(* IEC 61131-3 sources: CereveateHMI_Production_v2/CSharpBackend, 2 files *)

(* ---- FTP1_Simulation.st ---- *)
(* ============================================================
   FTP-1 POTLINE Simulation Program — FULL REPLACEMENT
   Auto-generated from Tag_master_Details_System_Upload.xlsx
   TOTAL TAGS: 128 (includes all 5 existing + 123 new)
   Set Sim_Enable := 1 to start, 0 to stop.
   Tags with NULL limits simulate within normal range only.
   All other tags oscillate across LL/HH -> triggers alarms.
   ============================================================ *)

VAR
    Sim_Enable  : BOOL := 0;

    (* --- Simulated tag variables --- *)
    PY1101A       : REAL := 1.16;
    Dir_PY1101A   : BOOL := 1;
    PY1101B       : REAL := 1.125;
    Dir_PY1101B   : BOOL := 1;
    PY1103A       : REAL := 17.45;
    Dir_PY1103A   : BOOL := 1;
    PY1103B       : REAL := 16.525;
    Dir_PY1103B   : BOOL := 1;
    TY1101A       : REAL := 59.4;
    Dir_TY1101A   : BOOL := 1;
    PY1104       : REAL := 7.35;
    Dir_PY1104   : BOOL := 1;
    PY1105A       : REAL := 0.405;
    Dir_PY1105A   : BOOL := 1;
    PY1105B       : REAL := 0.405;
    Dir_PY1105B   : BOOL := 1;
    PY1105C       : REAL := 0.405;
    Dir_PY1105C   : BOOL := 1;
    PY1105D       : REAL := 0.405;
    Dir_PY1105D   : BOOL := 1;
    PY1105E       : REAL := 0.405;
    Dir_PY1105E   : BOOL := 1;
    PY1105F       : REAL := 0.405;
    Dir_PY1105F   : BOOL := 1;
    PY1105G       : REAL := 0.405;
    Dir_PY1105G   : BOOL := 1;
    PY1105H       : REAL := 0.405;
    Dir_PY1105H   : BOOL := 1;
    PY1105I       : REAL := 0.405;
    Dir_PY1105I   : BOOL := 1;
    PY1105J       : REAL := 0.405;
    Dir_PY1105J   : BOOL := 1;
    TY1101B       : REAL := 75.0;
    Dir_TY1101B   : BOOL := 1;
    TY1101C       : REAL := 75.0;
    Dir_TY1101C   : BOOL := 1;
    TY1101D       : REAL := 75.0;
    Dir_TY1101D   : BOOL := 1;
    TY1101E       : REAL := 75.0;
    Dir_TY1101E   : BOOL := 1;
    TY1101F       : REAL := 75.0;
    Dir_TY1101F   : BOOL := 1;
    TY1101G       : REAL := 75.0;
    Dir_TY1101G   : BOOL := 1;
    TY1101H       : REAL := 75.0;
    Dir_TY1101H   : BOOL := 1;
    TY1102A       : REAL := 75.0;
    Dir_TY1102A   : BOOL := 1;
    TY1102B       : REAL := 75.0;
    Dir_TY1102B   : BOOL := 1;
    TY1102C       : REAL := 75.0;
    Dir_TY1102C   : BOOL := 1;
    TY1102D       : REAL := 75.0;
    Dir_TY1102D   : BOOL := 1;
    TY1102E       : REAL := 75.0;
    Dir_TY1102E   : BOOL := 1;
    TY1102F       : REAL := 75.0;
    Dir_TY1102F   : BOOL := 1;
    TY1102G       : REAL := 75.0;
    Dir_TY1102G   : BOOL := 1;
    TY1102H       : REAL := 75.0;
    Dir_TY1102H   : BOOL := 1;
    TY1103A       : REAL := 75.0;
    Dir_TY1103A   : BOOL := 1;
    TY1103B       : REAL := 75.0;
    Dir_TY1103B   : BOOL := 1;
    TY1103C       : REAL := 75.0;
    Dir_TY1103C   : BOOL := 1;
    TY1103D       : REAL := 75.0;
    Dir_TY1103D   : BOOL := 1;
    TY1103E       : REAL := 75.0;
    Dir_TY1103E   : BOOL := 1;
    TY1103F       : REAL := 75.0;
    Dir_TY1103F   : BOOL := 1;
    TY1103G       : REAL := 75.0;
    Dir_TY1103G   : BOOL := 1;
    TY1103H       : REAL := 75.0;
    Dir_TY1103H   : BOOL := 1;
    TY1104A       : REAL := 75.0;
    Dir_TY1104A   : BOOL := 1;
    TY1104B       : REAL := 75.0;
    Dir_TY1104B   : BOOL := 1;
    TY1104C       : REAL := 75.0;
    Dir_TY1104C   : BOOL := 1;
    TY1104D       : REAL := 75.0;
    Dir_TY1104D   : BOOL := 1;
    TY1104E       : REAL := 75.0;
    Dir_TY1104E   : BOOL := 1;
    TY1104F       : REAL := 75.0;
    Dir_TY1104F   : BOOL := 1;
    TY1104G       : REAL := 75.0;
    Dir_TY1104G   : BOOL := 1;
    TY1104H       : REAL := 75.0;
    Dir_TY1104H   : BOOL := 1;
    IYAN1101       : REAL := 45.0;
    Dir_IYAN1101   : BOOL := 1;
    IYAN1102       : REAL := 45.0;
    Dir_IYAN1102   : BOOL := 1;
    IYAN1103       : REAL := 45.0;
    Dir_IYAN1103   : BOOL := 1;
    IYAN1104       : REAL := 45.0;
    Dir_IYAN1104   : BOOL := 1;
    IYFBR1101       : REAL := 45.0;
    Dir_IYFBR1101   : BOOL := 1;
    IYFBR1102       : REAL := 45.0;
    Dir_IYFBR1102   : BOOL := 1;
    IYFBC1101       : REAL := 45.0;
    Dir_IYFBC1101   : BOOL := 1;
    IYFBC1102       : REAL := 45.0;
    Dir_IYFBC1102   : BOOL := 1;
    HZ1101A       : REAL := 50.0;
    Dir_HZ1101A   : BOOL := 1;
    HZ1102A       : REAL := 50.0;
    Dir_HZ1102A   : BOOL := 1;
    HZ1103A       : REAL := 50.0;
    Dir_HZ1103A   : BOOL := 1;
    HZ1104A       : REAL := 50.0;
    Dir_HZ1104A   : BOOL := 1;
    AY1101       : REAL := 42.5;
    Dir_AY1101   : BOOL := 1;
    AY1102       : REAL := 42.5;
    Dir_AY1102   : BOOL := 1;
    TY1105A       : REAL := 75.0;
    Dir_TY1105A   : BOOL := 1;
    TY1105B       : REAL := 75.0;
    Dir_TY1105B   : BOOL := 1;
    PDY1101       : REAL := 1.925;
    Dir_PDY1101   : BOOL := 1;
    PDY1102       : REAL := 1.925;
    Dir_PDY1102   : BOOL := 1;
    PDY1104       : REAL := 1.925;
    Dir_PDY1104   : BOOL := 1;
    PDY1105       : REAL := 1.925;
    Dir_PDY1105   : BOOL := 1;
    PDY1106A       : REAL := 1.925;
    Dir_PDY1106A   : BOOL := 1;
    PDY1107A       : REAL := 1.925;
    Dir_PDY1107A   : BOOL := 1;
    PDY1108       : REAL := 1.925;
    Dir_PDY1108   : BOOL := 1;
    PDY1109       : REAL := 1.925;
    Dir_PDY1109   : BOOL := 1;
    PDY1110       : REAL := 1.925;
    Dir_PDY1110   : BOOL := 1;
    FY1100       : REAL := 2250.0;
    Dir_FY1100   : BOOL := 1;
    VYAN1101A       : REAL := 3.75;
    Dir_VYAN1101A   : BOOL := 1;
    VYAN1101B       : REAL := 3.75;
    Dir_VYAN1101B   : BOOL := 1;
    VYAN1101C       : REAL := 3.75;
    Dir_VYAN1101C   : BOOL := 1;
    VYAN1101D       : REAL := 3.75;
    Dir_VYAN1101D   : BOOL := 1;
    VYAN1102A       : REAL := 3.75;
    Dir_VYAN1102A   : BOOL := 1;
    VYAN1102B       : REAL := 3.75;
    Dir_VYAN1102B   : BOOL := 1;
    VYAN1102C       : REAL := 3.75;
    Dir_VYAN1102C   : BOOL := 1;
    VYAN1102D       : REAL := 3.75;
    Dir_VYAN1102D   : BOOL := 1;
    VYAN1103A       : REAL := 3.75;
    Dir_VYAN1103A   : BOOL := 1;
    VYAN1103B       : REAL := 3.75;
    Dir_VYAN1103B   : BOOL := 1;
    VYAN1103C       : REAL := 3.75;
    Dir_VYAN1103C   : BOOL := 1;
    VYAN1103D       : REAL := 3.75;
    Dir_VYAN1103D   : BOOL := 1;
    VYAN1104A       : REAL := 3.75;
    Dir_VYAN1104A   : BOOL := 1;
    VYAN1104B       : REAL := 3.75;
    Dir_VYAN1104B   : BOOL := 1;
    VYAN1104C       : REAL := 3.75;
    Dir_VYAN1104C   : BOOL := 1;
    VYAN1104D       : REAL := 3.75;
    Dir_VYAN1104D   : BOOL := 1;
    PY1102A       : REAL := 22.5;
    Dir_PY1102A   : BOOL := 1;
    PY1102B       : REAL := 22.5;
    Dir_PY1102B   : BOOL := 1;
    PY1102C       : REAL := 22.5;
    Dir_PY1102C   : BOOL := 1;
    PY1102D       : REAL := 22.5;
    Dir_PY1102D   : BOOL := 1;
    LY3101       : REAL := 3.675;
    Dir_LY3101   : BOOL := 1;
    PY3101       : REAL := 1.925;
    Dir_PY3101   : BOOL := 1;
    LY1101       : REAL := 4.5;
    Dir_LY1101   : BOOL := 1;
    LY1102       : REAL := 4.5;
    Dir_LY1102   : BOOL := 1;
    FY3101       : REAL := 225.0;
    Dir_FY3101   : BOOL := 1;
    VY1101A       : REAL := 50.0;
    Dir_VY1101A   : BOOL := 1;
    FY1101       : REAL := 90.0;
    Dir_FY1101   : BOOL := 1;
    CV1101       : REAL := 52.5;
    Dir_CV1101   : BOOL := 1;
    TY3101       : REAL := 75.0;
    Dir_TY3101   : BOOL := 1;
    VYAN1101E       : REAL := 3.75;
    Dir_VYAN1101E   : BOOL := 1;
    VYAN1101F       : REAL := 3.75;
    Dir_VYAN1101F   : BOOL := 1;
    VYAN1101G       : REAL := 3.75;
    Dir_VYAN1101G   : BOOL := 1;
    VYAN1101H       : REAL := 3.75;
    Dir_VYAN1101H   : BOOL := 1;
    VYAN1102E       : REAL := 3.75;
    Dir_VYAN1102E   : BOOL := 1;
    VYAN1102F       : REAL := 3.75;
    Dir_VYAN1102F   : BOOL := 1;
    VYAN1102G       : REAL := 3.75;
    Dir_VYAN1102G   : BOOL := 1;
    VYAN1102H       : REAL := 3.75;
    Dir_VYAN1102H   : BOOL := 1;
    VYAN1103E       : REAL := 3.75;
    Dir_VYAN1103E   : BOOL := 1;
    VYAN1103F       : REAL := 3.75;
    Dir_VYAN1103F   : BOOL := 1;
    VYAN1103G       : REAL := 3.75;
    Dir_VYAN1103G   : BOOL := 1;
    VYAN1103H       : REAL := 3.75;
    Dir_VYAN1103H   : BOOL := 1;
    VYAN1104E       : REAL := 3.75;
    Dir_VYAN1104E   : BOOL := 1;
    VYAN1104F       : REAL := 3.75;
    Dir_VYAN1104F   : BOOL := 1;
    VYAN1104G       : REAL := 3.75;
    Dir_VYAN1104G   : BOOL := 1;
    VYAN1104H       : REAL := 3.75;
    Dir_VYAN1104H   : BOOL := 1;
    MV1101A       : REAL := 50.0;
    Dir_MV1101A   : BOOL := 1;
    MV1102A       : REAL := 50.0;
    Dir_MV1102A   : BOOL := 1;
    HZ1101B       : REAL := 50.0;
    Dir_HZ1101B   : BOOL := 1;
    HZ1102B       : REAL := 50.0;
    Dir_HZ1102B   : BOOL := 1;
    HZ1103B       : REAL := 50.0;
    Dir_HZ1103B   : BOOL := 1;
    HZ1104B       : REAL := 50.0;
    Dir_HZ1104B   : BOOL := 1;
    VT1101B       : REAL := 50.0;
    Dir_VT1101B   : BOOL := 1;
    CV1101B       : REAL := 52.5;
    Dir_CV1101B   : BOOL := 1;
    Fresh_SILO_MT       : REAL := 450.0;
    Dir_Fresh_SILO_MT   : BOOL := 1;
    Enrich_SILO_MT       : REAL := 450.0;
    Dir_Enrich_SILO_MT   : BOOL := 1;
END_VAR

(* ============================================================
   SIMULATION BODY
   ============================================================ *)
IF Sim_Enable THEN

    (* PY1101A - CHUTE SILO FAN OUTLET PRESSURE #1 [KPA] sim 0.48..1.84 *)
    IF Dir_PY1101A THEN
        PY1101A := PY1101A + 0.009067;
    ELSE
        PY1101A := PY1101A - 0.009067;
    END_IF;
    IF PY1101A >= 1.84 THEN Dir_PY1101A := 0; END_IF;
    IF PY1101A <= 0.48 THEN Dir_PY1101A := 1; END_IF;

    (* PY1101B - CHUTE SILO FAN OUTLET PRESSURE #2 [KPA] sim 0.64..1.61 *)
    IF Dir_PY1101B THEN
        PY1101B := PY1101B + 0.006467;
    ELSE
        PY1101B := PY1101B - 0.006467;
    END_IF;
    IF PY1101B >= 1.61 THEN Dir_PY1101B := 0; END_IF;
    IF PY1101B <= 0.64 THEN Dir_PY1101B := 1; END_IF;

    (* PY1103A - ID FAN OUTLET PRESSURE #1 [KPA] sim 9.6..25.3 *)
    IF Dir_PY1103A THEN
        PY1103A := PY1103A + 0.104667;
    ELSE
        PY1103A := PY1103A - 0.104667;
    END_IF;
    IF PY1103A >= 25.3 THEN Dir_PY1103A := 0; END_IF;
    IF PY1103A <= 9.6 THEN Dir_PY1103A := 1; END_IF;

    (* PY1103B - ID FAN OUTLET PRESSURE #2 [KPA] sim 11.2..21.85 *)
    IF Dir_PY1103B THEN
        PY1103B := PY1103B + 0.071;
    ELSE
        PY1103B := PY1103B - 0.071;
    END_IF;
    IF PY1103B >= 21.85 THEN Dir_PY1103B := 0; END_IF;
    IF PY1103B <= 11.2 THEN Dir_PY1103B := 1; END_IF;

    (* TY1101A - 1# ID FAN FRONT BEARING TEMPERATURE [°C] sim 36.0..82.8 *)
    IF Dir_TY1101A THEN
        TY1101A := TY1101A + 0.312;
    ELSE
        TY1101A := TY1101A - 0.312;
    END_IF;
    IF TY1101A >= 82.8 THEN Dir_TY1101A := 0; END_IF;
    IF TY1101A <= 36.0 THEN Dir_TY1101A := 1; END_IF;

    (* PY1104 - CHUTE  SILO FAN OUTLET OF PRESSURE [KPA] sim 3.2..11.5 *)
    IF Dir_PY1104 THEN
        PY1104 := PY1104 + 0.055333;
    ELSE
        PY1104 := PY1104 - 0.055333;
    END_IF;
    IF PY1104 >= 11.5 THEN Dir_PY1104 := 0; END_IF;
    IF PY1104 <= 3.2 THEN Dir_PY1104 := 1; END_IF;

    (* PY1105A - FILTER AIR BAG OF PRESSURE #1 [KPA] sim 0.12..0.69 *)
    IF Dir_PY1105A THEN
        PY1105A := PY1105A + 0.0038;
    ELSE
        PY1105A := PY1105A - 0.0038;
    END_IF;
    IF PY1105A >= 0.69 THEN Dir_PY1105A := 0; END_IF;
    IF PY1105A <= 0.12 THEN Dir_PY1105A := 1; END_IF;

    (* PY1105B - FILTER AIR BAG OF PRESSURE #2 [KPA] sim 0.12..0.69 *)
    IF Dir_PY1105B THEN
        PY1105B := PY1105B + 0.0038;
    ELSE
        PY1105B := PY1105B - 0.0038;
    END_IF;
    IF PY1105B >= 0.69 THEN Dir_PY1105B := 0; END_IF;
    IF PY1105B <= 0.12 THEN Dir_PY1105B := 1; END_IF;

    (* PY1105C - FILTER AIR BAG OF PRESSURE #3 [KPA] sim 0.12..0.69 *)
    IF Dir_PY1105C THEN
        PY1105C := PY1105C + 0.0038;
    ELSE
        PY1105C := PY1105C - 0.0038;
    END_IF;
    IF PY1105C >= 0.69 THEN Dir_PY1105C := 0; END_IF;
    IF PY1105C <= 0.12 THEN Dir_PY1105C := 1; END_IF;

    (* PY1105D - FILTER AIR BAG OF PRESSURE #4 [KPA] sim 0.12..0.69 *)
    IF Dir_PY1105D THEN
        PY1105D := PY1105D + 0.0038;
    ELSE
        PY1105D := PY1105D - 0.0038;
    END_IF;
    IF PY1105D >= 0.69 THEN Dir_PY1105D := 0; END_IF;
    IF PY1105D <= 0.12 THEN Dir_PY1105D := 1; END_IF;

    (* PY1105E - FILTER AIR BAG OF PRESSURE #5 [KPA] sim 0.12..0.69 *)
    IF Dir_PY1105E THEN
        PY1105E := PY1105E + 0.0038;
    ELSE
        PY1105E := PY1105E - 0.0038;
    END_IF;
    IF PY1105E >= 0.69 THEN Dir_PY1105E := 0; END_IF;
    IF PY1105E <= 0.12 THEN Dir_PY1105E := 1; END_IF;

    (* PY1105F - FILTER AIR BAG OF PRESSURE #6 [KPA] sim 0.12..0.69 *)
    IF Dir_PY1105F THEN
        PY1105F := PY1105F + 0.0038;
    ELSE
        PY1105F := PY1105F - 0.0038;
    END_IF;
    IF PY1105F >= 0.69 THEN Dir_PY1105F := 0; END_IF;
    IF PY1105F <= 0.12 THEN Dir_PY1105F := 1; END_IF;

    (* PY1105G - FILTER AIR BAG OF PRESSURE #7 [KPA] sim 0.12..0.69 *)
    IF Dir_PY1105G THEN
        PY1105G := PY1105G + 0.0038;
    ELSE
        PY1105G := PY1105G - 0.0038;
    END_IF;
    IF PY1105G >= 0.69 THEN Dir_PY1105G := 0; END_IF;
    IF PY1105G <= 0.12 THEN Dir_PY1105G := 1; END_IF;

    (* PY1105H - FILTER AIR BAG OF PRESSURE #8 [KPA] sim 0.12..0.69 *)
    IF Dir_PY1105H THEN
        PY1105H := PY1105H + 0.0038;
    ELSE
        PY1105H := PY1105H - 0.0038;
    END_IF;
    IF PY1105H >= 0.69 THEN Dir_PY1105H := 0; END_IF;
    IF PY1105H <= 0.12 THEN Dir_PY1105H := 1; END_IF;

    (* PY1105I - FILTER AIR BAG OF PRESSURE #9 [KPA] sim 0.12..0.69 *)
    IF Dir_PY1105I THEN
        PY1105I := PY1105I + 0.0038;
    ELSE
        PY1105I := PY1105I - 0.0038;
    END_IF;
    IF PY1105I >= 0.69 THEN Dir_PY1105I := 0; END_IF;
    IF PY1105I <= 0.12 THEN Dir_PY1105I := 1; END_IF;

    (* PY1105J - FILTER AIR BAG OF PRESSURE #10 [KPA] sim 0.12..0.69 *)
    IF Dir_PY1105J THEN
        PY1105J := PY1105J + 0.0038;
    ELSE
        PY1105J := PY1105J - 0.0038;
    END_IF;
    IF PY1105J >= 0.69 THEN Dir_PY1105J := 0; END_IF;
    IF PY1105J <= 0.12 THEN Dir_PY1105J := 1; END_IF;

    (* TY1101B - 1# ID FAN REAR BEARING TEMPERATURE [°C] sim 30.0..120.0 *)
    IF Dir_TY1101B THEN
        TY1101B := TY1101B + 0.6;
    ELSE
        TY1101B := TY1101B - 0.6;
    END_IF;
    IF TY1101B >= 120.0 THEN Dir_TY1101B := 0; END_IF;
    IF TY1101B <= 30.0 THEN Dir_TY1101B := 1; END_IF;

    (* TY1101C - 1# ID FAN MOTOR FRONT BEARING TEMPERATURE [°C] sim 30.0..120.0 *)
    IF Dir_TY1101C THEN
        TY1101C := TY1101C + 0.6;
    ELSE
        TY1101C := TY1101C - 0.6;
    END_IF;
    IF TY1101C >= 120.0 THEN Dir_TY1101C := 0; END_IF;
    IF TY1101C <= 30.0 THEN Dir_TY1101C := 1; END_IF;

    (* TY1101D - 1# ID FAN MOTOR REAR BEARING TEMPERATURE [°C] sim 30.0..120.0 *)
    IF Dir_TY1101D THEN
        TY1101D := TY1101D + 0.6;
    ELSE
        TY1101D := TY1101D - 0.6;
    END_IF;
    IF TY1101D >= 120.0 THEN Dir_TY1101D := 0; END_IF;
    IF TY1101D <= 30.0 THEN Dir_TY1101D := 1; END_IF;

    (* TY1101E - 1# ID FAN  MOTOR Winding temperature A [°C] sim 30.0..120.0 *)
    IF Dir_TY1101E THEN
        TY1101E := TY1101E + 0.6;
    ELSE
        TY1101E := TY1101E - 0.6;
    END_IF;
    IF TY1101E >= 120.0 THEN Dir_TY1101E := 0; END_IF;
    IF TY1101E <= 30.0 THEN Dir_TY1101E := 1; END_IF;

    (* TY1101F - 1# ID FAN  MOTOR Winding temperature B [°C] sim 30.0..120.0 *)
    IF Dir_TY1101F THEN
        TY1101F := TY1101F + 0.6;
    ELSE
        TY1101F := TY1101F - 0.6;
    END_IF;
    IF TY1101F >= 120.0 THEN Dir_TY1101F := 0; END_IF;
    IF TY1101F <= 30.0 THEN Dir_TY1101F := 1; END_IF;

    (* TY1101G - 1# ID FAN  MOTOR Winding temperature C [°C] sim 30.0..120.0 *)
    IF Dir_TY1101G THEN
        TY1101G := TY1101G + 0.6;
    ELSE
        TY1101G := TY1101G - 0.6;
    END_IF;
    IF TY1101G >= 120.0 THEN Dir_TY1101G := 0; END_IF;
    IF TY1101G <= 30.0 THEN Dir_TY1101G := 1; END_IF;

    (* TY1101H - 1# ID FAN INLET TEMPERATURE [°C] sim 30.0..120.0 *)
    IF Dir_TY1101H THEN
        TY1101H := TY1101H + 0.6;
    ELSE
        TY1101H := TY1101H - 0.6;
    END_IF;
    IF TY1101H >= 120.0 THEN Dir_TY1101H := 0; END_IF;
    IF TY1101H <= 30.0 THEN Dir_TY1101H := 1; END_IF;

    (* TY1102A - 2# ID FAN FRONT BEARING TEMPERATURE [°C] sim 30.0..120.0 *)
    IF Dir_TY1102A THEN
        TY1102A := TY1102A + 0.6;
    ELSE
        TY1102A := TY1102A - 0.6;
    END_IF;
    IF TY1102A >= 120.0 THEN Dir_TY1102A := 0; END_IF;
    IF TY1102A <= 30.0 THEN Dir_TY1102A := 1; END_IF;

    (* TY1102B - 2# ID FAN REAR BEARING TEMPERATURE [°C] sim 30.0..120.0 *)
    IF Dir_TY1102B THEN
        TY1102B := TY1102B + 0.6;
    ELSE
        TY1102B := TY1102B - 0.6;
    END_IF;
    IF TY1102B >= 120.0 THEN Dir_TY1102B := 0; END_IF;
    IF TY1102B <= 30.0 THEN Dir_TY1102B := 1; END_IF;

    (* TY1102C - 2# ID FAN MOTOR FRONT BEARING TEMPERATURE [°C] sim 30.0..120.0 *)
    IF Dir_TY1102C THEN
        TY1102C := TY1102C + 0.6;
    ELSE
        TY1102C := TY1102C - 0.6;
    END_IF;
    IF TY1102C >= 120.0 THEN Dir_TY1102C := 0; END_IF;
    IF TY1102C <= 30.0 THEN Dir_TY1102C := 1; END_IF;

    (* TY1102D - 2# ID FAN MOTOR REAR BEARING TEMPERATURE [°C] sim 30.0..120.0 *)
    IF Dir_TY1102D THEN
        TY1102D := TY1102D + 0.6;
    ELSE
        TY1102D := TY1102D - 0.6;
    END_IF;
    IF TY1102D >= 120.0 THEN Dir_TY1102D := 0; END_IF;
    IF TY1102D <= 30.0 THEN Dir_TY1102D := 1; END_IF;

    (* TY1102E - 2# ID FAN  MOTOR Winding temperature A [°C] sim 30.0..120.0 *)
    IF Dir_TY1102E THEN
        TY1102E := TY1102E + 0.6;
    ELSE
        TY1102E := TY1102E - 0.6;
    END_IF;
    IF TY1102E >= 120.0 THEN Dir_TY1102E := 0; END_IF;
    IF TY1102E <= 30.0 THEN Dir_TY1102E := 1; END_IF;

    (* TY1102F - 2# ID FAN  MOTOR Winding temperature B [°C] sim 30.0..120.0 *)
    IF Dir_TY1102F THEN
        TY1102F := TY1102F + 0.6;
    ELSE
        TY1102F := TY1102F - 0.6;
    END_IF;
    IF TY1102F >= 120.0 THEN Dir_TY1102F := 0; END_IF;
    IF TY1102F <= 30.0 THEN Dir_TY1102F := 1; END_IF;

    (* TY1102G - 2# ID FAN  MOTOR Winding temperature C [°C] sim 30.0..120.0 *)
    IF Dir_TY1102G THEN
        TY1102G := TY1102G + 0.6;
    ELSE
        TY1102G := TY1102G - 0.6;
    END_IF;
    IF TY1102G >= 120.0 THEN Dir_TY1102G := 0; END_IF;
    IF TY1102G <= 30.0 THEN Dir_TY1102G := 1; END_IF;

    (* TY1102H - 2# ID FAN INLET TEMPERATURE [°C] sim 30.0..120.0 *)
    IF Dir_TY1102H THEN
        TY1102H := TY1102H + 0.6;
    ELSE
        TY1102H := TY1102H - 0.6;
    END_IF;
    IF TY1102H >= 120.0 THEN Dir_TY1102H := 0; END_IF;
    IF TY1102H <= 30.0 THEN Dir_TY1102H := 1; END_IF;

    (* TY1103A - 3# ID FAN FRONT BEARING TEMPERATURE [°C] sim 30.0..120.0 *)
    IF Dir_TY1103A THEN
        TY1103A := TY1103A + 0.6;
    ELSE
        TY1103A := TY1103A - 0.6;
    END_IF;
    IF TY1103A >= 120.0 THEN Dir_TY1103A := 0; END_IF;
    IF TY1103A <= 30.0 THEN Dir_TY1103A := 1; END_IF;

    (* TY1103B - 3# ID FAN REAR BEARING TEMPERATURE [°C] sim 30.0..120.0 *)
    IF Dir_TY1103B THEN
        TY1103B := TY1103B + 0.6;
    ELSE
        TY1103B := TY1103B - 0.6;
    END_IF;
    IF TY1103B >= 120.0 THEN Dir_TY1103B := 0; END_IF;
    IF TY1103B <= 30.0 THEN Dir_TY1103B := 1; END_IF;

    (* TY1103C - 3# ID FAN MOTOR FRONT BEARING TEMPERATURE [°C] sim 30.0..120.0 *)
    IF Dir_TY1103C THEN
        TY1103C := TY1103C + 0.6;
    ELSE
        TY1103C := TY1103C - 0.6;
    END_IF;
    IF TY1103C >= 120.0 THEN Dir_TY1103C := 0; END_IF;
    IF TY1103C <= 30.0 THEN Dir_TY1103C := 1; END_IF;

    (* TY1103D - 3# ID FAN MOTOR REAR BEARING TEMPERATURE [°C] sim 30.0..120.0 *)
    IF Dir_TY1103D THEN
        TY1103D := TY1103D + 0.6;
    ELSE
        TY1103D := TY1103D - 0.6;
    END_IF;
    IF TY1103D >= 120.0 THEN Dir_TY1103D := 0; END_IF;
    IF TY1103D <= 30.0 THEN Dir_TY1103D := 1; END_IF;

    (* TY1103E - 3# ID FAN  MOTOR Winding temperature A [°C] sim 30.0..120.0 *)
    IF Dir_TY1103E THEN
        TY1103E := TY1103E + 0.6;
    ELSE
        TY1103E := TY1103E - 0.6;
    END_IF;
    IF TY1103E >= 120.0 THEN Dir_TY1103E := 0; END_IF;
    IF TY1103E <= 30.0 THEN Dir_TY1103E := 1; END_IF;

    (* TY1103F - 3# ID FAN  MOTOR Winding temperature B [°C] sim 30.0..120.0 *)
    IF Dir_TY1103F THEN
        TY1103F := TY1103F + 0.6;
    ELSE
        TY1103F := TY1103F - 0.6;
    END_IF;
    IF TY1103F >= 120.0 THEN Dir_TY1103F := 0; END_IF;
    IF TY1103F <= 30.0 THEN Dir_TY1103F := 1; END_IF;

    (* TY1103G - 3# ID FAN  MOTOR Winding temperature C [°C] sim 30.0..120.0 *)
    IF Dir_TY1103G THEN
        TY1103G := TY1103G + 0.6;
    ELSE
        TY1103G := TY1103G - 0.6;
    END_IF;
    IF TY1103G >= 120.0 THEN Dir_TY1103G := 0; END_IF;
    IF TY1103G <= 30.0 THEN Dir_TY1103G := 1; END_IF;

    (* TY1103H - 3# ID FAN INLET TEMPERATURE [°C] sim 30.0..120.0 *)
    IF Dir_TY1103H THEN
        TY1103H := TY1103H + 0.6;
    ELSE
        TY1103H := TY1103H - 0.6;
    END_IF;
    IF TY1103H >= 120.0 THEN Dir_TY1103H := 0; END_IF;
    IF TY1103H <= 30.0 THEN Dir_TY1103H := 1; END_IF;

    (* TY1104A - 4# ID FAN FRONT BEARING TEMPERATURE [°C] sim 30.0..120.0 *)
    IF Dir_TY1104A THEN
        TY1104A := TY1104A + 0.6;
    ELSE
        TY1104A := TY1104A - 0.6;
    END_IF;
    IF TY1104A >= 120.0 THEN Dir_TY1104A := 0; END_IF;
    IF TY1104A <= 30.0 THEN Dir_TY1104A := 1; END_IF;

    (* TY1104B - 4# ID FAN REAR BEARING TEMPERATURE [°C] sim 30.0..120.0 *)
    IF Dir_TY1104B THEN
        TY1104B := TY1104B + 0.6;
    ELSE
        TY1104B := TY1104B - 0.6;
    END_IF;
    IF TY1104B >= 120.0 THEN Dir_TY1104B := 0; END_IF;
    IF TY1104B <= 30.0 THEN Dir_TY1104B := 1; END_IF;

    (* TY1104C - 4# ID FAN MOTOR FRONT BEARING TEMPERATURE [°C] sim 30.0..120.0 *)
    IF Dir_TY1104C THEN
        TY1104C := TY1104C + 0.6;
    ELSE
        TY1104C := TY1104C - 0.6;
    END_IF;
    IF TY1104C >= 120.0 THEN Dir_TY1104C := 0; END_IF;
    IF TY1104C <= 30.0 THEN Dir_TY1104C := 1; END_IF;

    (* TY1104D - 4# ID FAN MOTOR REAR BEARING TEMPERATURE [°C] sim 30.0..120.0 *)
    IF Dir_TY1104D THEN
        TY1104D := TY1104D + 0.6;
    ELSE
        TY1104D := TY1104D - 0.6;
    END_IF;
    IF TY1104D >= 120.0 THEN Dir_TY1104D := 0; END_IF;
    IF TY1104D <= 30.0 THEN Dir_TY1104D := 1; END_IF;

    (* TY1104E - 4# ID FAN  MOTOR Winding temperature A [°C] sim 30.0..120.0 *)
    IF Dir_TY1104E THEN
        TY1104E := TY1104E + 0.6;
    ELSE
        TY1104E := TY1104E - 0.6;
    END_IF;
    IF TY1104E >= 120.0 THEN Dir_TY1104E := 0; END_IF;
    IF TY1104E <= 30.0 THEN Dir_TY1104E := 1; END_IF;

    (* TY1104F - 4# ID FAN  MOTOR Winding temperature B [°C] sim 30.0..120.0 *)
    IF Dir_TY1104F THEN
        TY1104F := TY1104F + 0.6;
    ELSE
        TY1104F := TY1104F - 0.6;
    END_IF;
    IF TY1104F >= 120.0 THEN Dir_TY1104F := 0; END_IF;
    IF TY1104F <= 30.0 THEN Dir_TY1104F := 1; END_IF;

    (* TY1104G - 4# ID FAN  MOTOR Winding temperature C [°C] sim 30.0..120.0 *)
    IF Dir_TY1104G THEN
        TY1104G := TY1104G + 0.6;
    ELSE
        TY1104G := TY1104G - 0.6;
    END_IF;
    IF TY1104G >= 120.0 THEN Dir_TY1104G := 0; END_IF;
    IF TY1104G <= 30.0 THEN Dir_TY1104G := 1; END_IF;

    (* TY1104H - 4# ID FAN INLET TEMPERATURE [°C] sim 30.0..120.0 *)
    IF Dir_TY1104H THEN
        TY1104H := TY1104H + 0.6;
    ELSE
        TY1104H := TY1104H - 0.6;
    END_IF;
    IF TY1104H >= 120.0 THEN Dir_TY1104H := 0; END_IF;
    IF TY1104H <= 30.0 THEN Dir_TY1104H := 1; END_IF;

    (* IYAN1101 - ID FAN CURRENT #1 [Amp] sim 10.0..80.0 *)
    IF Dir_IYAN1101 THEN
        IYAN1101 := IYAN1101 + 0.466667;
    ELSE
        IYAN1101 := IYAN1101 - 0.466667;
    END_IF;
    IF IYAN1101 >= 80.0 THEN Dir_IYAN1101 := 0; END_IF;
    IF IYAN1101 <= 10.0 THEN Dir_IYAN1101 := 1; END_IF;

    (* IYAN1102 - ID FAN CURRENT #2 [Amp] sim 10.0..80.0 *)
    IF Dir_IYAN1102 THEN
        IYAN1102 := IYAN1102 + 0.466667;
    ELSE
        IYAN1102 := IYAN1102 - 0.466667;
    END_IF;
    IF IYAN1102 >= 80.0 THEN Dir_IYAN1102 := 0; END_IF;
    IF IYAN1102 <= 10.0 THEN Dir_IYAN1102 := 1; END_IF;

    (* IYAN1103 - ID FAN CURRENT #3 [Amp] sim 10.0..80.0 *)
    IF Dir_IYAN1103 THEN
        IYAN1103 := IYAN1103 + 0.466667;
    ELSE
        IYAN1103 := IYAN1103 - 0.466667;
    END_IF;
    IF IYAN1103 >= 80.0 THEN Dir_IYAN1103 := 0; END_IF;
    IF IYAN1103 <= 10.0 THEN Dir_IYAN1103 := 1; END_IF;

    (* IYAN1104 - ID FAN CURRENT #4 [Amp] sim 10.0..80.0 *)
    IF Dir_IYAN1104 THEN
        IYAN1104 := IYAN1104 + 0.466667;
    ELSE
        IYAN1104 := IYAN1104 - 0.466667;
    END_IF;
    IF IYAN1104 >= 80.0 THEN Dir_IYAN1104 := 0; END_IF;
    IF IYAN1104 <= 10.0 THEN Dir_IYAN1104 := 1; END_IF;

    (* IYFBR1101 - ROOTS FAN CURRENT #1 [Amp] sim 10.0..80.0 *)
    IF Dir_IYFBR1101 THEN
        IYFBR1101 := IYFBR1101 + 0.466667;
    ELSE
        IYFBR1101 := IYFBR1101 - 0.466667;
    END_IF;
    IF IYFBR1101 >= 80.0 THEN Dir_IYFBR1101 := 0; END_IF;
    IF IYFBR1101 <= 10.0 THEN Dir_IYFBR1101 := 1; END_IF;

    (* IYFBR1102 - ROOTS FAN CURRENT #2 [Amp] sim 10.0..80.0 *)
    IF Dir_IYFBR1102 THEN
        IYFBR1102 := IYFBR1102 + 0.466667;
    ELSE
        IYFBR1102 := IYFBR1102 - 0.466667;
    END_IF;
    IF IYFBR1102 >= 80.0 THEN Dir_IYFBR1102 := 0; END_IF;
    IF IYFBR1102 <= 10.0 THEN Dir_IYFBR1102 := 1; END_IF;

    (* IYFBC1101 - HIGHT PRESSURE CENTRIFUGAL VENTILATOR #1 [Amp] sim 10.0..80.0 *)
    IF Dir_IYFBC1101 THEN
        IYFBC1101 := IYFBC1101 + 0.466667;
    ELSE
        IYFBC1101 := IYFBC1101 - 0.466667;
    END_IF;
    IF IYFBC1101 >= 80.0 THEN Dir_IYFBC1101 := 0; END_IF;
    IF IYFBC1101 <= 10.0 THEN Dir_IYFBC1101 := 1; END_IF;

    (* IYFBC1102 - HIGHT PRESSURE CENTRIFUGAL VENTILATOR #2 [Amp] sim 10.0..80.0 *)
    IF Dir_IYFBC1102 THEN
        IYFBC1102 := IYFBC1102 + 0.466667;
    ELSE
        IYFBC1102 := IYFBC1102 - 0.466667;
    END_IF;
    IF IYFBC1102 >= 80.0 THEN Dir_IYFBC1102 := 0; END_IF;
    IF IYFBC1102 <= 10.0 THEN Dir_IYFBC1102 := 1; END_IF;

    (* HZ1101A - ID FAN VALVE OF DEGREE (DAMPER FEEDBACK) #1 [%] sim 20.0..80.0 *)
    IF Dir_HZ1101A THEN
        HZ1101A := HZ1101A + 0.4;
    ELSE
        HZ1101A := HZ1101A - 0.4;
    END_IF;
    IF HZ1101A >= 80.0 THEN Dir_HZ1101A := 0; END_IF;
    IF HZ1101A <= 20.0 THEN Dir_HZ1101A := 1; END_IF;

    (* HZ1102A - ID FAN VALVE OF DEGREE (DAMPER FEEDBACK) #2 [%] sim 20.0..80.0 *)
    IF Dir_HZ1102A THEN
        HZ1102A := HZ1102A + 0.4;
    ELSE
        HZ1102A := HZ1102A - 0.4;
    END_IF;
    IF HZ1102A >= 80.0 THEN Dir_HZ1102A := 0; END_IF;
    IF HZ1102A <= 20.0 THEN Dir_HZ1102A := 1; END_IF;

    (* HZ1103A - ID FAN VALVE OF DEGREE (DAMPER FEEDBACK) #3 [%] sim 20.0..80.0 *)
    IF Dir_HZ1103A THEN
        HZ1103A := HZ1103A + 0.4;
    ELSE
        HZ1103A := HZ1103A - 0.4;
    END_IF;
    IF HZ1103A >= 80.0 THEN Dir_HZ1103A := 0; END_IF;
    IF HZ1103A <= 20.0 THEN Dir_HZ1103A := 1; END_IF;

    (* HZ1104A - ID FAN VALVE OF DEGREE (DAMPER FEEDBACK) #4 [%] sim 20.0..80.0 *)
    IF Dir_HZ1104A THEN
        HZ1104A := HZ1104A + 0.4;
    ELSE
        HZ1104A := HZ1104A - 0.4;
    END_IF;
    IF HZ1104A >= 80.0 THEN Dir_HZ1104A := 0; END_IF;
    IF HZ1104A <= 20.0 THEN Dir_HZ1104A := 1; END_IF;

    (* AY1101 - FTP-1 DUST ANALYZER [mg/m3] sim 5.0..80.0 *)
    IF Dir_AY1101 THEN
        AY1101 := AY1101 + 0.5;
    ELSE
        AY1101 := AY1101 - 0.5;
    END_IF;
    IF AY1101 >= 80.0 THEN Dir_AY1101 := 0; END_IF;
    IF AY1101 <= 5.0 THEN Dir_AY1101 := 1; END_IF;

    (* AY1102 - FTP-1 HF ANALYZER [mg/m3] sim 5.0..80.0 *)
    IF Dir_AY1102 THEN
        AY1102 := AY1102 + 0.5;
    ELSE
        AY1102 := AY1102 - 0.5;
    END_IF;
    IF AY1102 >= 80.0 THEN Dir_AY1102 := 0; END_IF;
    IF AY1102 <= 5.0 THEN Dir_AY1102 := 1; END_IF;

    (* TY1105A - FILTER INLET TEMPERATURE #1 [°C] sim 30.0..120.0 *)
    IF Dir_TY1105A THEN
        TY1105A := TY1105A + 0.6;
    ELSE
        TY1105A := TY1105A - 0.6;
    END_IF;
    IF TY1105A >= 120.0 THEN Dir_TY1105A := 0; END_IF;
    IF TY1105A <= 30.0 THEN Dir_TY1105A := 1; END_IF;

    (* TY1105B - FILTER INLET TEMPERATURE #2 [°C] sim 30.0..120.0 *)
    IF Dir_TY1105B THEN
        TY1105B := TY1105B + 0.6;
    ELSE
        TY1105B := TY1105B - 0.6;
    END_IF;
    IF TY1105B >= 120.0 THEN Dir_TY1105B := 0; END_IF;
    IF TY1105B <= 30.0 THEN Dir_TY1105B := 1; END_IF;

    (* PDY1101 - FILTER INLET  OUTLET PRESSURE #1 [KPA] sim 0.4..3.45 *)
    IF Dir_PDY1101 THEN
        PDY1101 := PDY1101 + 0.020333;
    ELSE
        PDY1101 := PDY1101 - 0.020333;
    END_IF;
    IF PDY1101 >= 3.45 THEN Dir_PDY1101 := 0; END_IF;
    IF PDY1101 <= 0.4 THEN Dir_PDY1101 := 1; END_IF;

    (* PDY1102 - FILTER INLET  OUTLET PRESSURE #2 [KPA] sim 0.4..3.45 *)
    IF Dir_PDY1102 THEN
        PDY1102 := PDY1102 + 0.020333;
    ELSE
        PDY1102 := PDY1102 - 0.020333;
    END_IF;
    IF PDY1102 >= 3.45 THEN Dir_PDY1102 := 0; END_IF;
    IF PDY1102 <= 0.4 THEN Dir_PDY1102 := 1; END_IF;

    (* PDY1104 - FILTER INLET  OUTLET PRESSURE #4 [KPA] sim 0.4..3.45 *)
    IF Dir_PDY1104 THEN
        PDY1104 := PDY1104 + 0.020333;
    ELSE
        PDY1104 := PDY1104 - 0.020333;
    END_IF;
    IF PDY1104 >= 3.45 THEN Dir_PDY1104 := 0; END_IF;
    IF PDY1104 <= 0.4 THEN Dir_PDY1104 := 1; END_IF;

    (* PDY1105 - FILTER INLET  OUTLET PRESSURE #5 [KPA] sim 0.4..3.45 *)
    IF Dir_PDY1105 THEN
        PDY1105 := PDY1105 + 0.020333;
    ELSE
        PDY1105 := PDY1105 - 0.020333;
    END_IF;
    IF PDY1105 >= 3.45 THEN Dir_PDY1105 := 0; END_IF;
    IF PDY1105 <= 0.4 THEN Dir_PDY1105 := 1; END_IF;

    (* PDY1106A - FILTER INLET  OUTLET PRESSURE #6 [KPA] sim 0.4..3.45 *)
    IF Dir_PDY1106A THEN
        PDY1106A := PDY1106A + 0.020333;
    ELSE
        PDY1106A := PDY1106A - 0.020333;
    END_IF;
    IF PDY1106A >= 3.45 THEN Dir_PDY1106A := 0; END_IF;
    IF PDY1106A <= 0.4 THEN Dir_PDY1106A := 1; END_IF;

    (* PDY1107A - FILTER INLET  OUTLET PRESSURE #7 [KPA] sim 0.4..3.45 *)
    IF Dir_PDY1107A THEN
        PDY1107A := PDY1107A + 0.020333;
    ELSE
        PDY1107A := PDY1107A - 0.020333;
    END_IF;
    IF PDY1107A >= 3.45 THEN Dir_PDY1107A := 0; END_IF;
    IF PDY1107A <= 0.4 THEN Dir_PDY1107A := 1; END_IF;

    (* PDY1108 - FILTER INLET  OUTLET PRESSURE #8 [KPA] sim 0.4..3.45 *)
    IF Dir_PDY1108 THEN
        PDY1108 := PDY1108 + 0.020333;
    ELSE
        PDY1108 := PDY1108 - 0.020333;
    END_IF;
    IF PDY1108 >= 3.45 THEN Dir_PDY1108 := 0; END_IF;
    IF PDY1108 <= 0.4 THEN Dir_PDY1108 := 1; END_IF;

    (* PDY1109 - FILTER INLET  OUTLET PRESSURE #9 [KPA] sim 0.4..3.45 *)
    IF Dir_PDY1109 THEN
        PDY1109 := PDY1109 + 0.020333;
    ELSE
        PDY1109 := PDY1109 - 0.020333;
    END_IF;
    IF PDY1109 >= 3.45 THEN Dir_PDY1109 := 0; END_IF;
    IF PDY1109 <= 0.4 THEN Dir_PDY1109 := 1; END_IF;

    (* PDY1110 - FILTER INLET  OUTLET PRESSURE #10 [KPA] sim 0.4..3.45 *)
    IF Dir_PDY1110 THEN
        PDY1110 := PDY1110 + 0.020333;
    ELSE
        PDY1110 := PDY1110 - 0.020333;
    END_IF;
    IF PDY1110 >= 3.45 THEN Dir_PDY1110 := 0; END_IF;
    IF PDY1110 <= 0.4 THEN Dir_PDY1110 := 1; END_IF;

    (* FY1100 - OUTLET FLOW [Nm3/Hr] sim 500.0..4000.0 *)
    IF Dir_FY1100 THEN
        FY1100 := FY1100 + 23.333333;
    ELSE
        FY1100 := FY1100 - 23.333333;
    END_IF;
    IF FY1100 >= 4000.0 THEN Dir_FY1100 := 0; END_IF;
    IF FY1100 <= 500.0 THEN Dir_FY1100 := 1; END_IF;

    (* VYAN1101A - ID FAN FRONT BEARING X VIBRATION #1 [mm/s] sim 0.5..7.0 *)
    IF Dir_VYAN1101A THEN
        VYAN1101A := VYAN1101A + 0.043333;
    ELSE
        VYAN1101A := VYAN1101A - 0.043333;
    END_IF;
    IF VYAN1101A >= 7.0 THEN Dir_VYAN1101A := 0; END_IF;
    IF VYAN1101A <= 0.5 THEN Dir_VYAN1101A := 1; END_IF;

    (* VYAN1101B - ID FAN FRONT BEARING Y VIBRATION #1 [mm/s] sim 0.5..7.0 *)
    IF Dir_VYAN1101B THEN
        VYAN1101B := VYAN1101B + 0.043333;
    ELSE
        VYAN1101B := VYAN1101B - 0.043333;
    END_IF;
    IF VYAN1101B >= 7.0 THEN Dir_VYAN1101B := 0; END_IF;
    IF VYAN1101B <= 0.5 THEN Dir_VYAN1101B := 1; END_IF;

    (* VYAN1101C - ID FAN REAR BEARING X VIBRATION #1 [mm/s] sim 0.5..7.0 *)
    IF Dir_VYAN1101C THEN
        VYAN1101C := VYAN1101C + 0.043333;
    ELSE
        VYAN1101C := VYAN1101C - 0.043333;
    END_IF;
    IF VYAN1101C >= 7.0 THEN Dir_VYAN1101C := 0; END_IF;
    IF VYAN1101C <= 0.5 THEN Dir_VYAN1101C := 1; END_IF;

    (* VYAN1101D - ID FAN REAR BEARING Y VIBRATION #1 [mm/s] sim 0.5..7.0 *)
    IF Dir_VYAN1101D THEN
        VYAN1101D := VYAN1101D + 0.043333;
    ELSE
        VYAN1101D := VYAN1101D - 0.043333;
    END_IF;
    IF VYAN1101D >= 7.0 THEN Dir_VYAN1101D := 0; END_IF;
    IF VYAN1101D <= 0.5 THEN Dir_VYAN1101D := 1; END_IF;

    (* VYAN1102A - ID FAN FRONT BEARING X VIBRATION #2 [mm/s] sim 0.5..7.0 *)
    IF Dir_VYAN1102A THEN
        VYAN1102A := VYAN1102A + 0.043333;
    ELSE
        VYAN1102A := VYAN1102A - 0.043333;
    END_IF;
    IF VYAN1102A >= 7.0 THEN Dir_VYAN1102A := 0; END_IF;
    IF VYAN1102A <= 0.5 THEN Dir_VYAN1102A := 1; END_IF;

    (* VYAN1102B - ID FAN FRONT BEARING Y VIBRATION #2 [mm/s] sim 0.5..7.0 *)
    IF Dir_VYAN1102B THEN
        VYAN1102B := VYAN1102B + 0.043333;
    ELSE
        VYAN1102B := VYAN1102B - 0.043333;
    END_IF;
    IF VYAN1102B >= 7.0 THEN Dir_VYAN1102B := 0; END_IF;
    IF VYAN1102B <= 0.5 THEN Dir_VYAN1102B := 1; END_IF;

    (* VYAN1102C - ID FAN REAR BEARING X VIBRATION #2 [mm/s] sim 0.5..7.0 *)
    IF Dir_VYAN1102C THEN
        VYAN1102C := VYAN1102C + 0.043333;
    ELSE
        VYAN1102C := VYAN1102C - 0.043333;
    END_IF;
    IF VYAN1102C >= 7.0 THEN Dir_VYAN1102C := 0; END_IF;
    IF VYAN1102C <= 0.5 THEN Dir_VYAN1102C := 1; END_IF;

    (* VYAN1102D - ID FAN REAR BEARING Y VIBRATION #2 [mm/s] sim 0.5..7.0 *)
    IF Dir_VYAN1102D THEN
        VYAN1102D := VYAN1102D + 0.043333;
    ELSE
        VYAN1102D := VYAN1102D - 0.043333;
    END_IF;
    IF VYAN1102D >= 7.0 THEN Dir_VYAN1102D := 0; END_IF;
    IF VYAN1102D <= 0.5 THEN Dir_VYAN1102D := 1; END_IF;

    (* VYAN1103A - ID FAN FRONT BEARING X VIBRATION #3 [mm/s] sim 0.5..7.0 *)
    IF Dir_VYAN1103A THEN
        VYAN1103A := VYAN1103A + 0.043333;
    ELSE
        VYAN1103A := VYAN1103A - 0.043333;
    END_IF;
    IF VYAN1103A >= 7.0 THEN Dir_VYAN1103A := 0; END_IF;
    IF VYAN1103A <= 0.5 THEN Dir_VYAN1103A := 1; END_IF;

    (* VYAN1103B - ID FAN FRONT BEARING Y VIBRATION #3 [mm/s] sim 0.5..7.0 *)
    IF Dir_VYAN1103B THEN
        VYAN1103B := VYAN1103B + 0.043333;
    ELSE
        VYAN1103B := VYAN1103B - 0.043333;
    END_IF;
    IF VYAN1103B >= 7.0 THEN Dir_VYAN1103B := 0; END_IF;
    IF VYAN1103B <= 0.5 THEN Dir_VYAN1103B := 1; END_IF;

    (* VYAN1103C - ID FAN REAR BEARING X VIBRATION #3 [mm/s] sim 0.5..7.0 *)
    IF Dir_VYAN1103C THEN
        VYAN1103C := VYAN1103C + 0.043333;
    ELSE
        VYAN1103C := VYAN1103C - 0.043333;
    END_IF;
    IF VYAN1103C >= 7.0 THEN Dir_VYAN1103C := 0; END_IF;
    IF VYAN1103C <= 0.5 THEN Dir_VYAN1103C := 1; END_IF;

    (* VYAN1103D - ID FAN REAR BEARING Y VIBRATION #3 [mm/s] sim 0.5..7.0 *)
    IF Dir_VYAN1103D THEN
        VYAN1103D := VYAN1103D + 0.043333;
    ELSE
        VYAN1103D := VYAN1103D - 0.043333;
    END_IF;
    IF VYAN1103D >= 7.0 THEN Dir_VYAN1103D := 0; END_IF;
    IF VYAN1103D <= 0.5 THEN Dir_VYAN1103D := 1; END_IF;

    (* VYAN1104A - ID FAN FRONT BEARING X VIBRATION #4 [mm/s] sim 0.5..7.0 *)
    IF Dir_VYAN1104A THEN
        VYAN1104A := VYAN1104A + 0.043333;
    ELSE
        VYAN1104A := VYAN1104A - 0.043333;
    END_IF;
    IF VYAN1104A >= 7.0 THEN Dir_VYAN1104A := 0; END_IF;
    IF VYAN1104A <= 0.5 THEN Dir_VYAN1104A := 1; END_IF;

    (* VYAN1104B - ID FAN FRONT BEARING Y VIBRATION #4 [mm/s] sim 0.5..7.0 *)
    IF Dir_VYAN1104B THEN
        VYAN1104B := VYAN1104B + 0.043333;
    ELSE
        VYAN1104B := VYAN1104B - 0.043333;
    END_IF;
    IF VYAN1104B >= 7.0 THEN Dir_VYAN1104B := 0; END_IF;
    IF VYAN1104B <= 0.5 THEN Dir_VYAN1104B := 1; END_IF;

    (* VYAN1104C - ID FAN REAR BEARING X VIBRATION #4 [mm/s] sim 0.5..7.0 *)
    IF Dir_VYAN1104C THEN
        VYAN1104C := VYAN1104C + 0.043333;
    ELSE
        VYAN1104C := VYAN1104C - 0.043333;
    END_IF;
    IF VYAN1104C >= 7.0 THEN Dir_VYAN1104C := 0; END_IF;
    IF VYAN1104C <= 0.5 THEN Dir_VYAN1104C := 1; END_IF;

    (* VYAN1104D - ID FAN REAR BEARING Y VIBRATION #4 [mm/s] sim 0.5..7.0 *)
    IF Dir_VYAN1104D THEN
        VYAN1104D := VYAN1104D + 0.043333;
    ELSE
        VYAN1104D := VYAN1104D - 0.043333;
    END_IF;
    IF VYAN1104D >= 7.0 THEN Dir_VYAN1104D := 0; END_IF;
    IF VYAN1104D <= 0.5 THEN Dir_VYAN1104D := 1; END_IF;

    (* PY1102A - ID FAN INLET PRESSURE #1 [KPA] sim 5.0..40.0 *)
    IF Dir_PY1102A THEN
        PY1102A := PY1102A + 0.233333;
    ELSE
        PY1102A := PY1102A - 0.233333;
    END_IF;
    IF PY1102A >= 40.0 THEN Dir_PY1102A := 0; END_IF;
    IF PY1102A <= 5.0 THEN Dir_PY1102A := 1; END_IF;

    (* PY1102B - ID FAN INLET PRESSURE #2 [KPA] sim 5.0..40.0 *)
    IF Dir_PY1102B THEN
        PY1102B := PY1102B + 0.233333;
    ELSE
        PY1102B := PY1102B - 0.233333;
    END_IF;
    IF PY1102B >= 40.0 THEN Dir_PY1102B := 0; END_IF;
    IF PY1102B <= 5.0 THEN Dir_PY1102B := 1; END_IF;

    (* PY1102C - ID FAN INLET PRESSURE #3 [KPA] sim 5.0..40.0 *)
    IF Dir_PY1102C THEN
        PY1102C := PY1102C + 0.233333;
    ELSE
        PY1102C := PY1102C - 0.233333;
    END_IF;
    IF PY1102C >= 40.0 THEN Dir_PY1102C := 0; END_IF;
    IF PY1102C <= 5.0 THEN Dir_PY1102C := 1; END_IF;

    (* PY1102D - ID FAN INLET PRESSURE #4 [KPA] sim 5.0..40.0 *)
    IF Dir_PY1102D THEN
        PY1102D := PY1102D + 0.233333;
    ELSE
        PY1102D := PY1102D - 0.233333;
    END_IF;
    IF PY1102D >= 40.0 THEN Dir_PY1102D := 0; END_IF;
    IF PY1102D <= 5.0 THEN Dir_PY1102D := 1; END_IF;

    (* LY3101 - CYCLE TANK LEVEL DETECTE [M] sim 1.6..5.75 *)
    IF Dir_LY3101 THEN
        LY3101 := LY3101 + 0.027667;
    ELSE
        LY3101 := LY3101 - 0.027667;
    END_IF;
    IF LY3101 >= 5.75 THEN Dir_LY3101 := 0; END_IF;
    IF LY3101 <= 1.6 THEN Dir_LY3101 := 1; END_IF;

    (* PY3101 - CYCLE OUTLET PIPE PRESSURE [KPA] sim 0.4..3.45 *)
    IF Dir_PY3101 THEN
        PY3101 := PY3101 + 0.020333;
    ELSE
        PY3101 := PY3101 - 0.020333;
    END_IF;
    IF PY3101 >= 3.45 THEN Dir_PY3101 := 0; END_IF;
    IF PY3101 <= 0.4 THEN Dir_PY3101 := 1; END_IF;

    (* LY1101 - FRESH ALUMINA CANBIN LEVEL [M] sim 1.0..8.0 *)
    IF Dir_LY1101 THEN
        LY1101 := LY1101 + 0.046667;
    ELSE
        LY1101 := LY1101 - 0.046667;
    END_IF;
    IF LY1101 >= 8.0 THEN Dir_LY1101 := 0; END_IF;
    IF LY1101 <= 1.0 THEN Dir_LY1101 := 1; END_IF;

    (* LY1102 - ENRICH ALUMINA CABIN LEVEL  [M] sim 1.0..8.0 *)
    IF Dir_LY1102 THEN
        LY1102 := LY1102 + 0.046667;
    ELSE
        LY1102 := LY1102 - 0.046667;
    END_IF;
    IF LY1102 >= 8.0 THEN Dir_LY1102 := 0; END_IF;
    IF LY1102 <= 1.0 THEN Dir_LY1102 := 1; END_IF;

    (* FY3101 - CYCLE OUTLET PIPE FLOW METER [m3/h] sim 50.0..400.0 *)
    IF Dir_FY3101 THEN
        FY3101 := FY3101 + 2.333333;
    ELSE
        FY3101 := FY3101 - 2.333333;
    END_IF;
    IF FY3101 >= 400.0 THEN Dir_FY3101 := 0; END_IF;
    IF FY3101 <= 50.0 THEN Dir_FY3101 := 1; END_IF;

    (* VY1101A - FRONT VALVE  DEGREE OF DESSLAGGING [%] sim 20.0..80.0 *)
    IF Dir_VY1101A THEN
        VY1101A := VY1101A + 0.4;
    ELSE
        VY1101A := VY1101A - 0.4;
    END_IF;
    IF VY1101A >= 80.0 THEN Dir_VY1101A := 0; END_IF;
    IF VY1101A <= 20.0 THEN Dir_VY1101A := 1; END_IF;

    (* FY1101 - FRESH ALUMINA FLOW [Ton/h] sim 20.0..160.0 *)
    IF Dir_FY1101 THEN
        FY1101 := FY1101 + 0.933333;
    ELSE
        FY1101 := FY1101 - 0.933333;
    END_IF;
    IF FY1101 >= 160.0 THEN Dir_FY1101 := 0; END_IF;
    IF FY1101 <= 20.0 THEN Dir_FY1101 := 1; END_IF;

    (* CV1101 - FRENQUENCE OF Fresh alumina silo bottom screw conveyor [Hz] sim 50.0..55.0 *)
    IF Dir_CV1101 THEN
        CV1101 := CV1101 + 0.033333;
    ELSE
        CV1101 := CV1101 - 0.033333;
    END_IF;
    IF CV1101 >= 55.0 THEN Dir_CV1101 := 0; END_IF;
    IF CV1101 <= 50.0 THEN Dir_CV1101 := 1; END_IF;

    (* TY3101 - CYCLE WATER OUTLET TEMPERATURE [°C] sim 30.0..120.0 *)
    IF Dir_TY3101 THEN
        TY3101 := TY3101 + 0.6;
    ELSE
        TY3101 := TY3101 - 0.6;
    END_IF;
    IF TY3101 >= 120.0 THEN Dir_TY3101 := 0; END_IF;
    IF TY3101 <= 30.0 THEN Dir_TY3101 := 1; END_IF;

    (* VYAN1101E - ID FAN MOTOR FRONT BEARING X VIBRATION #1 [mm/s] sim 0.5..7.0 *)
    IF Dir_VYAN1101E THEN
        VYAN1101E := VYAN1101E + 0.043333;
    ELSE
        VYAN1101E := VYAN1101E - 0.043333;
    END_IF;
    IF VYAN1101E >= 7.0 THEN Dir_VYAN1101E := 0; END_IF;
    IF VYAN1101E <= 0.5 THEN Dir_VYAN1101E := 1; END_IF;

    (* VYAN1101F - ID FAN MOTOR FRONT BEARING Y VIBRATION #1 [mm/s] sim 0.5..7.0 *)
    IF Dir_VYAN1101F THEN
        VYAN1101F := VYAN1101F + 0.043333;
    ELSE
        VYAN1101F := VYAN1101F - 0.043333;
    END_IF;
    IF VYAN1101F >= 7.0 THEN Dir_VYAN1101F := 0; END_IF;
    IF VYAN1101F <= 0.5 THEN Dir_VYAN1101F := 1; END_IF;

    (* VYAN1101G - ID FAN MOTOR  REAR BEARING X VIBRATION #1 [mm/s] sim 0.5..7.0 *)
    IF Dir_VYAN1101G THEN
        VYAN1101G := VYAN1101G + 0.043333;
    ELSE
        VYAN1101G := VYAN1101G - 0.043333;
    END_IF;
    IF VYAN1101G >= 7.0 THEN Dir_VYAN1101G := 0; END_IF;
    IF VYAN1101G <= 0.5 THEN Dir_VYAN1101G := 1; END_IF;

    (* VYAN1101H - ID FAN MOTOR REAR BEARING Y VIBRATION #1 [mm/s] sim 0.5..7.0 *)
    IF Dir_VYAN1101H THEN
        VYAN1101H := VYAN1101H + 0.043333;
    ELSE
        VYAN1101H := VYAN1101H - 0.043333;
    END_IF;
    IF VYAN1101H >= 7.0 THEN Dir_VYAN1101H := 0; END_IF;
    IF VYAN1101H <= 0.5 THEN Dir_VYAN1101H := 1; END_IF;

    (* VYAN1102E - ID FAN MOTOR FRONT BEARING X VIBRATION #2 [mm/s] sim 0.5..7.0 *)
    IF Dir_VYAN1102E THEN
        VYAN1102E := VYAN1102E + 0.043333;
    ELSE
        VYAN1102E := VYAN1102E - 0.043333;
    END_IF;
    IF VYAN1102E >= 7.0 THEN Dir_VYAN1102E := 0; END_IF;
    IF VYAN1102E <= 0.5 THEN Dir_VYAN1102E := 1; END_IF;

    (* VYAN1102F - ID FAN MOTOR FRONT BEARING Y VIBRATION #2 [mm/s] sim 0.5..7.0 *)
    IF Dir_VYAN1102F THEN
        VYAN1102F := VYAN1102F + 0.043333;
    ELSE
        VYAN1102F := VYAN1102F - 0.043333;
    END_IF;
    IF VYAN1102F >= 7.0 THEN Dir_VYAN1102F := 0; END_IF;
    IF VYAN1102F <= 0.5 THEN Dir_VYAN1102F := 1; END_IF;

    (* VYAN1102G - ID FAN MOTOR  REAR BEARING X VIBRATION #2 [mm/s] sim 0.5..7.0 *)
    IF Dir_VYAN1102G THEN
        VYAN1102G := VYAN1102G + 0.043333;
    ELSE
        VYAN1102G := VYAN1102G - 0.043333;
    END_IF;
    IF VYAN1102G >= 7.0 THEN Dir_VYAN1102G := 0; END_IF;
    IF VYAN1102G <= 0.5 THEN Dir_VYAN1102G := 1; END_IF;

    (* VYAN1102H - ID FAN MOTOR REAR BEARING Y VIBRATION #2 [mm/s] sim 0.5..7.0 *)
    IF Dir_VYAN1102H THEN
        VYAN1102H := VYAN1102H + 0.043333;
    ELSE
        VYAN1102H := VYAN1102H - 0.043333;
    END_IF;
    IF VYAN1102H >= 7.0 THEN Dir_VYAN1102H := 0; END_IF;
    IF VYAN1102H <= 0.5 THEN Dir_VYAN1102H := 1; END_IF;

    (* VYAN1103E - ID FAN MOTOR FRONT BEARING X VIBRATION #3 [mm/s] sim 0.5..7.0 *)
    IF Dir_VYAN1103E THEN
        VYAN1103E := VYAN1103E + 0.043333;
    ELSE
        VYAN1103E := VYAN1103E - 0.043333;
    END_IF;
    IF VYAN1103E >= 7.0 THEN Dir_VYAN1103E := 0; END_IF;
    IF VYAN1103E <= 0.5 THEN Dir_VYAN1103E := 1; END_IF;

    (* VYAN1103F - ID FAN MOTOR FRONT BEARING Y VIBRATION #3 [mm/s] sim 0.5..7.0 *)
    IF Dir_VYAN1103F THEN
        VYAN1103F := VYAN1103F + 0.043333;
    ELSE
        VYAN1103F := VYAN1103F - 0.043333;
    END_IF;
    IF VYAN1103F >= 7.0 THEN Dir_VYAN1103F := 0; END_IF;
    IF VYAN1103F <= 0.5 THEN Dir_VYAN1103F := 1; END_IF;

    (* VYAN1103G - ID FAN MOTOR  REAR BEARING X VIBRATION #3 [mm/s] sim 0.5..7.0 *)
    IF Dir_VYAN1103G THEN
        VYAN1103G := VYAN1103G + 0.043333;
    ELSE
        VYAN1103G := VYAN1103G - 0.043333;
    END_IF;
    IF VYAN1103G >= 7.0 THEN Dir_VYAN1103G := 0; END_IF;
    IF VYAN1103G <= 0.5 THEN Dir_VYAN1103G := 1; END_IF;

    (* VYAN1103H - ID FAN MOTOR REAR BEARING Y VIBRATION #3 [mm/s] sim 0.5..7.0 *)
    IF Dir_VYAN1103H THEN
        VYAN1103H := VYAN1103H + 0.043333;
    ELSE
        VYAN1103H := VYAN1103H - 0.043333;
    END_IF;
    IF VYAN1103H >= 7.0 THEN Dir_VYAN1103H := 0; END_IF;
    IF VYAN1103H <= 0.5 THEN Dir_VYAN1103H := 1; END_IF;

    (* VYAN1104E - ID FAN MOTOR FRONT BEARING X VIBRATION #4 [mm/s] sim 0.5..7.0 *)
    IF Dir_VYAN1104E THEN
        VYAN1104E := VYAN1104E + 0.043333;
    ELSE
        VYAN1104E := VYAN1104E - 0.043333;
    END_IF;
    IF VYAN1104E >= 7.0 THEN Dir_VYAN1104E := 0; END_IF;
    IF VYAN1104E <= 0.5 THEN Dir_VYAN1104E := 1; END_IF;

    (* VYAN1104F - ID FAN MOTOR FRONT BEARING Y VIBRATION #4 [mm/s] sim 0.5..7.0 *)
    IF Dir_VYAN1104F THEN
        VYAN1104F := VYAN1104F + 0.043333;
    ELSE
        VYAN1104F := VYAN1104F - 0.043333;
    END_IF;
    IF VYAN1104F >= 7.0 THEN Dir_VYAN1104F := 0; END_IF;
    IF VYAN1104F <= 0.5 THEN Dir_VYAN1104F := 1; END_IF;

    (* VYAN1104G - ID FAN MOTOR  REAR BEARING X VIBRATION #4 [mm/s] sim 0.5..7.0 *)
    IF Dir_VYAN1104G THEN
        VYAN1104G := VYAN1104G + 0.043333;
    ELSE
        VYAN1104G := VYAN1104G - 0.043333;
    END_IF;
    IF VYAN1104G >= 7.0 THEN Dir_VYAN1104G := 0; END_IF;
    IF VYAN1104G <= 0.5 THEN Dir_VYAN1104G := 1; END_IF;

    (* VYAN1104H - ID FAN MOTOR REAR BEARING Y VIBRATION #4 [mm/s] sim 0.5..7.0 *)
    IF Dir_VYAN1104H THEN
        VYAN1104H := VYAN1104H + 0.043333;
    ELSE
        VYAN1104H := VYAN1104H - 0.043333;
    END_IF;
    IF VYAN1104H >= 7.0 THEN Dir_VYAN1104H := 0; END_IF;
    IF VYAN1104H <= 0.5 THEN Dir_VYAN1104H := 1; END_IF;

    (* MV1101A - Feedback of the regulating damper for cold air valve No.1 of the main flue [%] sim 20.0..80.0 *)
    IF Dir_MV1101A THEN
        MV1101A := MV1101A + 0.4;
    ELSE
        MV1101A := MV1101A - 0.4;
    END_IF;
    IF MV1101A >= 80.0 THEN Dir_MV1101A := 0; END_IF;
    IF MV1101A <= 20.0 THEN Dir_MV1101A := 1; END_IF;

    (* MV1102A - Feedback of the regulating damper for cold air valve No.2 of the main flue [%] sim 20.0..80.0 *)
    IF Dir_MV1102A THEN
        MV1102A := MV1102A + 0.4;
    ELSE
        MV1102A := MV1102A - 0.4;
    END_IF;
    IF MV1102A >= 80.0 THEN Dir_MV1102A := 0; END_IF;
    IF MV1102A <= 20.0 THEN Dir_MV1102A := 1; END_IF;

    (* HZ1101B - ID FAN REGULAR VALVE COMMAND #1 [%] sim 20.0..80.0 *)
    IF Dir_HZ1101B THEN
        HZ1101B := HZ1101B + 0.4;
    ELSE
        HZ1101B := HZ1101B - 0.4;
    END_IF;
    IF HZ1101B >= 80.0 THEN Dir_HZ1101B := 0; END_IF;
    IF HZ1101B <= 20.0 THEN Dir_HZ1101B := 1; END_IF;

    (* HZ1102B - ID FAN REGULAR VALVE COMMAND #2 [%] sim 20.0..80.0 *)
    IF Dir_HZ1102B THEN
        HZ1102B := HZ1102B + 0.4;
    ELSE
        HZ1102B := HZ1102B - 0.4;
    END_IF;
    IF HZ1102B >= 80.0 THEN Dir_HZ1102B := 0; END_IF;
    IF HZ1102B <= 20.0 THEN Dir_HZ1102B := 1; END_IF;

    (* HZ1103B - ID FAN REGULAR VALVE COMMAND #3 [%] sim 20.0..80.0 *)
    IF Dir_HZ1103B THEN
        HZ1103B := HZ1103B + 0.4;
    ELSE
        HZ1103B := HZ1103B - 0.4;
    END_IF;
    IF HZ1103B >= 80.0 THEN Dir_HZ1103B := 0; END_IF;
    IF HZ1103B <= 20.0 THEN Dir_HZ1103B := 1; END_IF;

    (* HZ1104B - ID FAN REGULAR VALVE COMMAND #4 [%] sim 20.0..80.0 *)
    IF Dir_HZ1104B THEN
        HZ1104B := HZ1104B + 0.4;
    ELSE
        HZ1104B := HZ1104B - 0.4;
    END_IF;
    IF HZ1104B >= 80.0 THEN Dir_HZ1104B := 0; END_IF;
    IF HZ1104B <= 20.0 THEN Dir_HZ1104B := 1; END_IF;

    (* VT1101B - SETPOINT OF THE FRESH STORAGE TANK REGULATING VALVE [%] sim 20.0..80.0 *)
    IF Dir_VT1101B THEN
        VT1101B := VT1101B + 0.4;
    ELSE
        VT1101B := VT1101B - 0.4;
    END_IF;
    IF VT1101B >= 80.0 THEN Dir_VT1101B := 0; END_IF;
    IF VT1101B <= 20.0 THEN Dir_VT1101B := 1; END_IF;

    (* CV1101B - SETPOINT OF Fresh alumina silo bottom screw conveyor [Hz] sim 50.0..55.0 *)
    IF Dir_CV1101B THEN
        CV1101B := CV1101B + 0.033333;
    ELSE
        CV1101B := CV1101B - 0.033333;
    END_IF;
    IF CV1101B >= 55.0 THEN Dir_CV1101B := 0; END_IF;
    IF CV1101B <= 50.0 THEN Dir_CV1101B := 1; END_IF;

    (* Fresh_SILO_MT - PRIMARY SILO LEVEL IN MT [MT] sim 100.0..800.0 *)
    IF Dir_Fresh_SILO_MT THEN
        Fresh_SILO_MT := Fresh_SILO_MT + 4.666667;
    ELSE
        Fresh_SILO_MT := Fresh_SILO_MT - 4.666667;
    END_IF;
    IF Fresh_SILO_MT >= 800.0 THEN Dir_Fresh_SILO_MT := 0; END_IF;
    IF Fresh_SILO_MT <= 100.0 THEN Dir_Fresh_SILO_MT := 1; END_IF;

    (* Enrich_SILO_MT - ENRICH SILO LEVEL IN MT [MT] sim 100.0..800.0 *)
    IF Dir_Enrich_SILO_MT THEN
        Enrich_SILO_MT := Enrich_SILO_MT + 4.666667;
    ELSE
        Enrich_SILO_MT := Enrich_SILO_MT - 4.666667;
    END_IF;
    IF Enrich_SILO_MT >= 800.0 THEN Dir_Enrich_SILO_MT := 0; END_IF;
    IF Enrich_SILO_MT <= 100.0 THEN Dir_Enrich_SILO_MT := 1; END_IF;

END_IF;

(* ---- FTP1_ST_Body.st ---- *)
(* ----------------------------------------------------
 * FTP-1 POTLINE Simulation
 * Same pattern as welding sim: one sim_step, SIN-based
 * Runs in main task. Set Sim_Enable := 1 to activate.
 * ----------------------------------------------------*)

IF Sim_Enable THEN

    (* Advance shared angle — same as welding sim_step *)
    sim_step := sim_step + 0.07;
    IF sim_step > 6.28 THEN sim_step := 0.0; END_IF;

    (* PY1101A [KPA] base=1.135 ±0.5938 range 0.51..1.76 *)
    PY1101A := 1.135 + (SIN(sim_step + 0.0) * 0.5938);

    (* PY1101B [KPA] base=1.11 ±0.4085 range 0.68..1.54 *)
    PY1101B := 1.11 + (SIN(sim_step + 0.39) * 0.4085);

    (* PY1103A [KPA] base=17.2 ±6.65 range 10.2..24.2 *)
    PY1103A := 17.2 + (SIN(sim_step + 0.78) * 6.65);

    (* PY1103B [KPA] base=16.4 ±4.275 range 11.9..20.9 *)
    PY1103B := 16.4 + (SIN(sim_step + 1.17) * 4.275);

    (* TY1101A [°C] base=58.725 ±19.4513 range 38.25..79.2 *)
    TY1101A := 58.725 + (SIN(sim_step + 1.56) * 19.4513);

    (* PY1104 [KPA] base=7.2 ±3.61 range 3.4..11.0 *)
    PY1104 := 7.2 + (SIN(sim_step + 1.95) * 3.61);

    (* PY1105A [KPA] base=0.3938 ±0.2529 range 0.1275..0.66 *)
    PY1105A := 0.3938 + (SIN(sim_step + 2.34) * 0.2529);

    (* PY1105B [KPA] base=0.3938 ±0.2529 range 0.1275..0.66 *)
    PY1105B := 0.3938 + (SIN(sim_step + 2.73) * 0.2529);

    (* PY1105C [KPA] base=0.3938 ±0.2529 range 0.1275..0.66 *)
    PY1105C := 0.3938 + (SIN(sim_step + 3.12) * 0.2529);

    (* PY1105D [KPA] base=0.3938 ±0.2529 range 0.1275..0.66 *)
    PY1105D := 0.3938 + (SIN(sim_step + 3.51) * 0.2529);

    (* PY1105E [KPA] base=0.3938 ±0.2529 range 0.1275..0.66 *)
    PY1105E := 0.3938 + (SIN(sim_step + 3.9) * 0.2529);

    (* PY1105F [KPA] base=0.3938 ±0.2529 range 0.1275..0.66 *)
    PY1105F := 0.3938 + (SIN(sim_step + 4.29) * 0.2529);

    (* PY1105G [KPA] base=0.3938 ±0.2529 range 0.1275..0.66 *)
    PY1105G := 0.3938 + (SIN(sim_step + 4.68) * 0.2529);

    (* PY1105H [KPA] base=0.3938 ±0.2529 range 0.1275..0.66 *)
    PY1105H := 0.3938 + (SIN(sim_step + 5.07) * 0.2529);

    (* PY1105I [KPA] base=0.3938 ±0.2529 range 0.1275..0.66 *)
    PY1105I := 0.3938 + (SIN(sim_step + 5.46) * 0.2529);

    (* PY1105J [KPA] base=0.3938 ±0.2529 range 0.1275..0.66 *)
    PY1105J := 0.3938 + (SIN(sim_step + 5.85) * 0.2529);

    (* TY1101B [°C] base=75.0 ±42.75 range 30.0..120.0 *)
    TY1101B := 75.0 + (SIN(sim_step + 0.0) * 42.75);

    (* TY1101C [°C] base=75.0 ±42.75 range 30.0..120.0 *)
    TY1101C := 75.0 + (SIN(sim_step + 0.39) * 42.75);

    (* TY1101D [°C] base=75.0 ±42.75 range 30.0..120.0 *)
    TY1101D := 75.0 + (SIN(sim_step + 0.78) * 42.75);

    (* TY1101E [°C] base=75.0 ±42.75 range 30.0..120.0 *)
    TY1101E := 75.0 + (SIN(sim_step + 1.17) * 42.75);

    (* TY1101F [°C] base=75.0 ±42.75 range 30.0..120.0 *)
    TY1101F := 75.0 + (SIN(sim_step + 1.56) * 42.75);

    (* TY1101G [°C] base=75.0 ±42.75 range 30.0..120.0 *)
    TY1101G := 75.0 + (SIN(sim_step + 1.95) * 42.75);

    (* TY1101H [°C] base=75.0 ±42.75 range 30.0..120.0 *)
    TY1101H := 75.0 + (SIN(sim_step + 2.34) * 42.75);

    (* TY1102A [°C] base=75.0 ±42.75 range 30.0..120.0 *)
    TY1102A := 75.0 + (SIN(sim_step + 2.73) * 42.75);

    (* TY1102B [°C] base=75.0 ±42.75 range 30.0..120.0 *)
    TY1102B := 75.0 + (SIN(sim_step + 3.12) * 42.75);

    (* TY1102C [°C] base=75.0 ±42.75 range 30.0..120.0 *)
    TY1102C := 75.0 + (SIN(sim_step + 3.51) * 42.75);

    (* TY1102D [°C] base=75.0 ±42.75 range 30.0..120.0 *)
    TY1102D := 75.0 + (SIN(sim_step + 3.9) * 42.75);

    (* TY1102E [°C] base=75.0 ±42.75 range 30.0..120.0 *)
    TY1102E := 75.0 + (SIN(sim_step + 4.29) * 42.75);

    (* TY1102F [°C] base=75.0 ±42.75 range 30.0..120.0 *)
    TY1102F := 75.0 + (SIN(sim_step + 4.68) * 42.75);

    (* TY1102G [°C] base=75.0 ±42.75 range 30.0..120.0 *)
    TY1102G := 75.0 + (SIN(sim_step + 5.07) * 42.75);

    (* TY1102H [°C] base=75.0 ±42.75 range 30.0..120.0 *)
    TY1102H := 75.0 + (SIN(sim_step + 5.46) * 42.75);

    (* TY1103A [°C] base=75.0 ±42.75 range 30.0..120.0 *)
    TY1103A := 75.0 + (SIN(sim_step + 5.85) * 42.75);

    (* TY1103B [°C] base=75.0 ±42.75 range 30.0..120.0 *)
    TY1103B := 75.0 + (SIN(sim_step + 0.0) * 42.75);

    (* TY1103C [°C] base=75.0 ±42.75 range 30.0..120.0 *)
    TY1103C := 75.0 + (SIN(sim_step + 0.39) * 42.75);

    (* TY1103D [°C] base=75.0 ±42.75 range 30.0..120.0 *)
    TY1103D := 75.0 + (SIN(sim_step + 0.78) * 42.75);

    (* TY1103E [°C] base=75.0 ±42.75 range 30.0..120.0 *)
    TY1103E := 75.0 + (SIN(sim_step + 1.17) * 42.75);

    (* TY1103F [°C] base=75.0 ±42.75 range 30.0..120.0 *)
    TY1103F := 75.0 + (SIN(sim_step + 1.56) * 42.75);

    (* TY1103G [°C] base=75.0 ±42.75 range 30.0..120.0 *)
    TY1103G := 75.0 + (SIN(sim_step + 1.95) * 42.75);

    (* TY1103H [°C] base=75.0 ±42.75 range 30.0..120.0 *)
    TY1103H := 75.0 + (SIN(sim_step + 2.34) * 42.75);

    (* TY1104A [°C] base=75.0 ±42.75 range 30.0..120.0 *)
    TY1104A := 75.0 + (SIN(sim_step + 2.73) * 42.75);

    (* TY1104B [°C] base=75.0 ±42.75 range 30.0..120.0 *)
    TY1104B := 75.0 + (SIN(sim_step + 3.12) * 42.75);

    (* TY1104C [°C] base=75.0 ±42.75 range 30.0..120.0 *)
    TY1104C := 75.0 + (SIN(sim_step + 3.51) * 42.75);

    (* TY1104D [°C] base=75.0 ±42.75 range 30.0..120.0 *)
    TY1104D := 75.0 + (SIN(sim_step + 3.9) * 42.75);

    (* TY1104E [°C] base=75.0 ±42.75 range 30.0..120.0 *)
    TY1104E := 75.0 + (SIN(sim_step + 4.29) * 42.75);

    (* TY1104F [°C] base=75.0 ±42.75 range 30.0..120.0 *)
    TY1104F := 75.0 + (SIN(sim_step + 4.68) * 42.75);

    (* TY1104G [°C] base=75.0 ±42.75 range 30.0..120.0 *)
    TY1104G := 75.0 + (SIN(sim_step + 5.07) * 42.75);

    (* TY1104H [°C] base=75.0 ±42.75 range 30.0..120.0 *)
    TY1104H := 75.0 + (SIN(sim_step + 5.46) * 42.75);

    (* IYAN1101 [Amp] base=45.0 ±33.25 range 10.0..80.0 *)
    IYAN1101 := 45.0 + (SIN(sim_step + 5.85) * 33.25);

    (* IYAN1102 [Amp] base=45.0 ±33.25 range 10.0..80.0 *)
    IYAN1102 := 45.0 + (SIN(sim_step + 0.0) * 33.25);

    (* IYAN1103 [Amp] base=45.0 ±33.25 range 10.0..80.0 *)
    IYAN1103 := 45.0 + (SIN(sim_step + 0.39) * 33.25);

    (* IYAN1104 [Amp] base=45.0 ±33.25 range 10.0..80.0 *)
    IYAN1104 := 45.0 + (SIN(sim_step + 0.78) * 33.25);

    (* IYFBR1101 [Amp] base=45.0 ±33.25 range 10.0..80.0 *)
    IYFBR1101 := 45.0 + (SIN(sim_step + 1.17) * 33.25);

    (* IYFBR1102 [Amp] base=45.0 ±33.25 range 10.0..80.0 *)
    IYFBR1102 := 45.0 + (SIN(sim_step + 1.56) * 33.25);

    (* IYFBC1101 [Amp] base=45.0 ±33.25 range 10.0..80.0 *)
    IYFBC1101 := 45.0 + (SIN(sim_step + 1.95) * 33.25);

    (* IYFBC1102 [Amp] base=45.0 ±33.25 range 10.0..80.0 *)
    IYFBC1102 := 45.0 + (SIN(sim_step + 2.34) * 33.25);

    (* HZ1101A [%] base=50.0 ±28.5 range 20.0..80.0 *)
    HZ1101A := 50.0 + (SIN(sim_step + 2.73) * 28.5);

    (* HZ1102A [%] base=50.0 ±28.5 range 20.0..80.0 *)
    HZ1102A := 50.0 + (SIN(sim_step + 3.12) * 28.5);

    (* HZ1103A [%] base=50.0 ±28.5 range 20.0..80.0 *)
    HZ1103A := 50.0 + (SIN(sim_step + 3.51) * 28.5);

    (* HZ1104A [%] base=50.0 ±28.5 range 20.0..80.0 *)
    HZ1104A := 50.0 + (SIN(sim_step + 3.9) * 28.5);

    (* AY1101 [mg/m3] base=42.5 ±35.625 range 5.0..80.0 *)
    AY1101 := 42.5 + (SIN(sim_step + 4.29) * 35.625);

    (* AY1102 [mg/m3] base=42.5 ±35.625 range 5.0..80.0 *)
    AY1102 := 42.5 + (SIN(sim_step + 4.68) * 35.625);

    (* TY1105A [°C] base=75.0 ±42.75 range 30.0..120.0 *)
    TY1105A := 75.0 + (SIN(sim_step + 5.07) * 42.75);

    (* TY1105B [°C] base=75.0 ±42.75 range 30.0..120.0 *)
    TY1105B := 75.0 + (SIN(sim_step + 5.46) * 42.75);

    (* PDY1101 [KPA] base=1.8625 ±1.3656 range 0.425..3.3 *)
    PDY1101 := 1.8625 + (SIN(sim_step + 5.85) * 1.3656);

    (* PDY1102 [KPA] base=1.8625 ±1.3656 range 0.425..3.3 *)
    PDY1102 := 1.8625 + (SIN(sim_step + 0.0) * 1.3656);

    (* PDY1104 [KPA] base=1.8625 ±1.3656 range 0.425..3.3 *)
    PDY1104 := 1.8625 + (SIN(sim_step + 0.39) * 1.3656);

    (* PDY1105 [KPA] base=1.8625 ±1.3656 range 0.425..3.3 *)
    PDY1105 := 1.8625 + (SIN(sim_step + 0.78) * 1.3656);

    (* PDY1106A [KPA] base=1.8625 ±1.3656 range 0.425..3.3 *)
    PDY1106A := 1.8625 + (SIN(sim_step + 1.17) * 1.3656);

    (* PDY1107A [KPA] base=1.8625 ±1.3656 range 0.425..3.3 *)
    PDY1107A := 1.8625 + (SIN(sim_step + 1.56) * 1.3656);

    (* PDY1108 [KPA] base=1.8625 ±1.3656 range 0.425..3.3 *)
    PDY1108 := 1.8625 + (SIN(sim_step + 1.95) * 1.3656);

    (* PDY1109 [KPA] base=1.8625 ±1.3656 range 0.425..3.3 *)
    PDY1109 := 1.8625 + (SIN(sim_step + 2.34) * 1.3656);

    (* PDY1110 [KPA] base=1.8625 ±1.3656 range 0.425..3.3 *)
    PDY1110 := 1.8625 + (SIN(sim_step + 2.73) * 1.3656);

    (* FY1100 [Nm3/Hr] base=2250.0 ±1662.5 range 500.0..4000.0 *)
    FY1100 := 2250.0 + (SIN(sim_step + 3.12) * 1662.5);

    (* VYAN1101A [mm/s] base=3.75 ±3.0875 range 0.5..7.0 *)
    VYAN1101A := 3.75 + (SIN(sim_step + 3.51) * 3.0875);

    (* VYAN1101B [mm/s] base=3.75 ±3.0875 range 0.5..7.0 *)
    VYAN1101B := 3.75 + (SIN(sim_step + 3.9) * 3.0875);

    (* VYAN1101C [mm/s] base=3.75 ±3.0875 range 0.5..7.0 *)
    VYAN1101C := 3.75 + (SIN(sim_step + 4.29) * 3.0875);

    (* VYAN1101D [mm/s] base=3.75 ±3.0875 range 0.5..7.0 *)
    VYAN1101D := 3.75 + (SIN(sim_step + 4.68) * 3.0875);

    (* VYAN1102A [mm/s] base=3.75 ±3.0875 range 0.5..7.0 *)
    VYAN1102A := 3.75 + (SIN(sim_step + 5.07) * 3.0875);

    (* VYAN1102B [mm/s] base=3.75 ±3.0875 range 0.5..7.0 *)
    VYAN1102B := 3.75 + (SIN(sim_step + 5.46) * 3.0875);

    (* VYAN1102C [mm/s] base=3.75 ±3.0875 range 0.5..7.0 *)
    VYAN1102C := 3.75 + (SIN(sim_step + 5.85) * 3.0875);

    (* VYAN1102D [mm/s] base=3.75 ±3.0875 range 0.5..7.0 *)
    VYAN1102D := 3.75 + (SIN(sim_step + 0.0) * 3.0875);

    (* VYAN1103A [mm/s] base=3.75 ±3.0875 range 0.5..7.0 *)
    VYAN1103A := 3.75 + (SIN(sim_step + 0.39) * 3.0875);

    (* VYAN1103B [mm/s] base=3.75 ±3.0875 range 0.5..7.0 *)
    VYAN1103B := 3.75 + (SIN(sim_step + 0.78) * 3.0875);

    (* VYAN1103C [mm/s] base=3.75 ±3.0875 range 0.5..7.0 *)
    VYAN1103C := 3.75 + (SIN(sim_step + 1.17) * 3.0875);

    (* VYAN1103D [mm/s] base=3.75 ±3.0875 range 0.5..7.0 *)
    VYAN1103D := 3.75 + (SIN(sim_step + 1.56) * 3.0875);

    (* VYAN1104A [mm/s] base=3.75 ±3.0875 range 0.5..7.0 *)
    VYAN1104A := 3.75 + (SIN(sim_step + 1.95) * 3.0875);

    (* VYAN1104B [mm/s] base=3.75 ±3.0875 range 0.5..7.0 *)
    VYAN1104B := 3.75 + (SIN(sim_step + 2.34) * 3.0875);

    (* VYAN1104C [mm/s] base=3.75 ±3.0875 range 0.5..7.0 *)
    VYAN1104C := 3.75 + (SIN(sim_step + 2.73) * 3.0875);

    (* VYAN1104D [mm/s] base=3.75 ±3.0875 range 0.5..7.0 *)
    VYAN1104D := 3.75 + (SIN(sim_step + 3.12) * 3.0875);

    (* PY1102A [KPA] base=22.5 ±16.625 range 5.0..40.0 *)
    PY1102A := 22.5 + (SIN(sim_step + 3.51) * 16.625);

    (* PY1102B [KPA] base=22.5 ±16.625 range 5.0..40.0 *)
    PY1102B := 22.5 + (SIN(sim_step + 3.9) * 16.625);

    (* PY1102C [KPA] base=22.5 ±16.625 range 5.0..40.0 *)
    PY1102C := 22.5 + (SIN(sim_step + 4.29) * 16.625);

    (* PY1102D [KPA] base=22.5 ±16.625 range 5.0..40.0 *)
    PY1102D := 22.5 + (SIN(sim_step + 4.68) * 16.625);

    (* LY3101 [M] base=3.6 ±1.805 range 1.7..5.5 *)
    LY3101 := 3.6 + (SIN(sim_step + 5.07) * 1.805);

    (* PY3101 [KPA] base=1.8625 ±1.3656 range 0.425..3.3 *)
    PY3101 := 1.8625 + (SIN(sim_step + 5.46) * 1.3656);

    (* LY1101 [M] base=4.5 ±3.325 range 1.0..8.0 *)
    LY1101 := 4.5 + (SIN(sim_step + 5.85) * 3.325);

    (* LY1102 [M] base=4.5 ±3.325 range 1.0..8.0 *)
    LY1102 := 4.5 + (SIN(sim_step + 0.0) * 3.325);

    (* FY3101 [m3/h] base=225.0 ±166.25 range 50.0..400.0 *)
    FY3101 := 225.0 + (SIN(sim_step + 0.39) * 166.25);

    (* VY1101A [%] base=50.0 ±28.5 range 20.0..80.0 *)
    VY1101A := 50.0 + (SIN(sim_step + 0.78) * 28.5);

    (* FY1101 [Ton/h] base=90.0 ±66.5 range 20.0..160.0 *)
    FY1101 := 90.0 + (SIN(sim_step + 1.17) * 66.5);

    (* CV1101 [Hz] base=52.5 ±2.375 range 50.0..55.0 *)
    CV1101 := 52.5 + (SIN(sim_step + 1.56) * 2.375);

    (* TY3101 [°C] base=75.0 ±42.75 range 30.0..120.0 *)
    TY3101 := 75.0 + (SIN(sim_step + 1.95) * 42.75);

    (* VYAN1101E [mm/s] base=3.75 ±3.0875 range 0.5..7.0 *)
    VYAN1101E := 3.75 + (SIN(sim_step + 2.34) * 3.0875);

    (* VYAN1101F [mm/s] base=3.75 ±3.0875 range 0.5..7.0 *)
    VYAN1101F := 3.75 + (SIN(sim_step + 2.73) * 3.0875);

    (* VYAN1101G [mm/s] base=3.75 ±3.0875 range 0.5..7.0 *)
    VYAN1101G := 3.75 + (SIN(sim_step + 3.12) * 3.0875);

    (* VYAN1101H [mm/s] base=3.75 ±3.0875 range 0.5..7.0 *)
    VYAN1101H := 3.75 + (SIN(sim_step + 3.51) * 3.0875);

    (* VYAN1102E [mm/s] base=3.75 ±3.0875 range 0.5..7.0 *)
    VYAN1102E := 3.75 + (SIN(sim_step + 3.9) * 3.0875);

    (* VYAN1102F [mm/s] base=3.75 ±3.0875 range 0.5..7.0 *)
    VYAN1102F := 3.75 + (SIN(sim_step + 4.29) * 3.0875);

    (* VYAN1102G [mm/s] base=3.75 ±3.0875 range 0.5..7.0 *)
    VYAN1102G := 3.75 + (SIN(sim_step + 4.68) * 3.0875);

    (* VYAN1102H [mm/s] base=3.75 ±3.0875 range 0.5..7.0 *)
    VYAN1102H := 3.75 + (SIN(sim_step + 5.07) * 3.0875);

    (* VYAN1103E [mm/s] base=3.75 ±3.0875 range 0.5..7.0 *)
    VYAN1103E := 3.75 + (SIN(sim_step + 5.46) * 3.0875);

    (* VYAN1103F [mm/s] base=3.75 ±3.0875 range 0.5..7.0 *)
    VYAN1103F := 3.75 + (SIN(sim_step + 5.85) * 3.0875);

    (* VYAN1103G [mm/s] base=3.75 ±3.0875 range 0.5..7.0 *)
    VYAN1103G := 3.75 + (SIN(sim_step + 0.0) * 3.0875);

    (* VYAN1103H [mm/s] base=3.75 ±3.0875 range 0.5..7.0 *)
    VYAN1103H := 3.75 + (SIN(sim_step + 0.39) * 3.0875);

    (* VYAN1104E [mm/s] base=3.75 ±3.0875 range 0.5..7.0 *)
    VYAN1104E := 3.75 + (SIN(sim_step + 0.78) * 3.0875);

    (* VYAN1104F [mm/s] base=3.75 ±3.0875 range 0.5..7.0 *)
    VYAN1104F := 3.75 + (SIN(sim_step + 1.17) * 3.0875);

    (* VYAN1104G [mm/s] base=3.75 ±3.0875 range 0.5..7.0 *)
    VYAN1104G := 3.75 + (SIN(sim_step + 1.56) * 3.0875);

    (* VYAN1104H [mm/s] base=3.75 ±3.0875 range 0.5..7.0 *)
    VYAN1104H := 3.75 + (SIN(sim_step + 1.95) * 3.0875);

    (* MV1101A [%] base=50.0 ±28.5 range 20.0..80.0 *)
    MV1101A := 50.0 + (SIN(sim_step + 2.34) * 28.5);

    (* MV1102A [%] base=50.0 ±28.5 range 20.0..80.0 *)
    MV1102A := 50.0 + (SIN(sim_step + 2.73) * 28.5);

    (* HZ1101B [%] base=50.0 ±28.5 range 20.0..80.0 *)
    HZ1101B := 50.0 + (SIN(sim_step + 3.12) * 28.5);

    (* HZ1102B [%] base=50.0 ±28.5 range 20.0..80.0 *)
    HZ1102B := 50.0 + (SIN(sim_step + 3.51) * 28.5);

    (* HZ1103B [%] base=50.0 ±28.5 range 20.0..80.0 *)
    HZ1103B := 50.0 + (SIN(sim_step + 3.9) * 28.5);

    (* HZ1104B [%] base=50.0 ±28.5 range 20.0..80.0 *)
    HZ1104B := 50.0 + (SIN(sim_step + 4.29) * 28.5);

    (* VT1101B [%] base=50.0 ±28.5 range 20.0..80.0 *)
    VT1101B := 50.0 + (SIN(sim_step + 4.68) * 28.5);

    (* CV1101B [Hz] base=52.5 ±2.375 range 50.0..55.0 *)
    CV1101B := 52.5 + (SIN(sim_step + 5.07) * 2.375);

    (* Fresh_SILO_MT [MT] base=450.0 ±332.5 range 100.0..800.0 *)
    Fresh_SILO_MT := 450.0 + (SIN(sim_step + 5.46) * 332.5);

    (* Enrich_SILO_MT [MT] base=450.0 ±332.5 range 100.0..800.0 *)
    Enrich_SILO_MT := 450.0 + (SIN(sim_step + 5.85) * 332.5);

ELSE

    (* Sim OFF — reset step only, keep last values *)
    sim_step := 0.0;

END_IF;
